// TwinCAT 3 PLC project LoggingHelper
// Title: Logging Helper
// Company: Beckhoff Industrial
// ProjectVersion: 0.1.0
// ProgramVersion: 3.1.4026.22
// libraries:
//   Tc2_Standard, * (Beckhoff Automation GmbH)
//   Tc2_System, * (Beckhoff Automation GmbH)
//   Tc2_Utilities, * (Beckhoff Automation GmbH)
// project tree:
//   Loggers/Interfaces/ I_LocalLogger.TcIO, I_Logger.TcIO
//   Loggers/ LocalLogger.TcPOU
//   LogMessages/Interfaces/ I_LogSource.TcIO, I_LogMessage.TcIO, I_LogArgument.TcIO
//   LogMessages/ LogMessage.TcPOU, LogSource.TcPOU
//   / Parameters.TcGVL, PlcTask.TcTTO
//   Project Information/ F_GetCompany.TcPOU, F_GetTitle.TcPOU, F_GetVersion.TcPOU
//   SimpleLogger/ I_LogPublisher.TcIO, LogHelper.TcPOU
//   Version/ Global_Version.TcGVL
//   _Internal/Interfaces/ I_Base.TcIO

CONFIGURATION LoggingHelper
    RESOURCE PLC ON TwinCAT3
        TASK PlcTask(INTERVAL := T#10ms, PRIORITY := 20);
    END_RESOURCE
END_CONFIGURATION

// ---- Parameters.TcGVL
{attribute 'qualified_only'}
VAR_GLOBAL CONSTANT
	MaxMessages : USINT := 10;
END_VAR

// ---- Version/Global_Version.TcGVL
{attribute 'TcGenerated'}
{attribute 'no-analysis'}
{attribute 'linkalways'}
// This function has been automatically generated from the project information.
VAR_GLOBAL CONSTANT
	{attribute 'const_non_replaced'}
	stLibVersion_Logging_Helper : ST_LibVersion := (iMajor := 0, iMinor := 1, iBuild := 0, iRevision := 0, nFlags := 0, sVersion := '0.1.0');
END_VAR

// ---- Loggers/Interfaces/I_LocalLogger.TcIO
INTERFACE I_LocalLogger EXTENDS I_Logger

METHOD ClearLog
VAR_INPUT
END_VAR
END_METHOD

{attribute 'monitoring' := 'call'}
PROPERTY Messages : REFERENCE TO ARRAY[0..Parameters.MaxMessages - 1] OF T_MaxString
GET
END_GET
END_PROPERTY

END_INTERFACE

// ---- Loggers/Interfaces/I_Logger.TcIO
INTERFACE I_Logger EXTENDS I_Base

METHOD LogMessage
VAR_INPUT
	Source	 : I_LogSource;
	Message	 : I_LogMessage;
	Argument : I_LogArgument := 0;
END_VAR
END_METHOD

END_INTERFACE

// ---- LogMessages/Interfaces/I_LogSource.TcIO
INTERFACE I_LogSource EXTENDS I_Base

{attribute 'monitoring':='call'}
PROPERTY SourceName : T_MaxString
GET
END_GET
END_PROPERTY

{attribute 'monitoring':='call'}
PROPERTY Timestamp : T_FILETIME64
GET
END_GET
END_PROPERTY

END_INTERFACE

// ---- LogMessages/Interfaces/I_LogMessage.TcIO
INTERFACE I_LogMessage EXTENDS I_Base

{attribute 'monitoring':='call'}
PROPERTY Message : T_MaxString
GET
END_GET
END_PROPERTY

{attribute 'monitoring':='call'}
PROPERTY Severity : USINT
GET
END_GET
END_PROPERTY

END_INTERFACE

// ---- LogMessages/Interfaces/I_LogArgument.TcIO
INTERFACE I_LogArgument EXTENDS I_Base

METHOD ToString : T_MaxString
VAR_INPUT
END_VAR
END_METHOD

END_INTERFACE

// ---- SimpleLogger/I_LogPublisher.TcIO
INTERFACE I_LogPublisher EXTENDS I_Base

METHOD Subscribe : BOOL
VAR_INPUT
	Logger : I_Logger;
END_VAR
END_METHOD

METHOD Unsubscribe : BOOL
VAR_INPUT
	Logger : I_Logger;
END_VAR
END_METHOD

END_INTERFACE

// ---- _Internal/Interfaces/I_Base.TcIO
INTERFACE I_Base EXTENDS SYSTEM.__QUERYINTERFACE

END_INTERFACE

// ---- Loggers/LocalLogger.TcPOU
FUNCTION_BLOCK LocalLogger IMPLEMENTS I_LocalLogger
VAR
	{attribute 'hide'}
	_Messages	 : ARRAY[0..Parameters.MaxMessages - 1] OF T_MaxString;
END_VAR

METHOD ClearLog
VAR_INPUT
END_VAR
VAR
	i : UDINT;
END_VAR
FOR i := 0 TO Parameters.MaxMessages - 1 DO
	_Messages[i] := '';
END_FOR
END_METHOD

METHOD LogMessage
VAR_INPUT
	Source	 : I_LogSource;
	Message	 : I_LogMessage;
	Argument : I_LogArgument := 0;
END_VAR

VAR
	TimeStamp  : T_FILETIME64;
	TimeString : T_MaxString;
	i : UDINT;
END_VAR
IF Source.TimeStamp = 0 THEN
	TimeStamp := F_GetSystemTime();
ELSE
	TimeStamp := Source.Timestamp;
END_IF

TimeString := SYSTEMTIME_TO_STRING(FILETIME64_TO_SYSTEMTIME(TimeStamp));
//shift messages down
FOR i := 2 TO Parameters.MaxMessages - 1 DO
	_Messages[Parameters.MaxMessages - i] := _Messages[Parameters.MaxMessages - 1 - i];
END_FOR

_Messages[0] := CONCAT(TimeString, CONCAT(' ', CONCAT(Source.SourceName, CONCAT(': ', Message.Message))));
IF Argument <> 0 THEN
	_Messages[0] := CONCAT(_Messages[0], CONCAT(' : ', Argument.ToString()));
END_IF
END_METHOD

{attribute 'monitoring' := 'call'}
PROPERTY Messages : REFERENCE TO ARRAY[0..Parameters.MaxMessages - 1] OF T_MaxString
GET
Messages REF= _Messages;
END_GET
END_PROPERTY

END_FUNCTION_BLOCK

// ---- LogMessages/LogMessage.TcPOU
FUNCTION_BLOCK LogMessage IMPLEMENTS I_LogMessage
VAR
	{attribute 'hide'}
	_Message : T_MaxString;
	{attribute 'hide'}
	_Severity : USINT;
END_VAR

{attribute 'monitoring':='call'}
PROPERTY Message : T_MaxString
GET
Message := _Message;
END_GET
SET
_Message := Message;
END_SET
END_PROPERTY

{attribute 'monitoring':='call'}
PROPERTY Severity : USINT
GET
Severity := _Severity;
END_GET
SET
_Severity := Severity;
END_SET
END_PROPERTY

END_FUNCTION_BLOCK

// ---- LogMessages/LogSource.TcPOU
FUNCTION_BLOCK LogSource IMPLEMENTS I_LogSource
VAR
	{attribute 'hide'}
	_SourceName : T_MaxString;
	{attribute 'hide'}
	_Timestamp : T_FILETIME64;
END_VAR

{attribute 'monitoring':='call'}
PROPERTY SourceName : T_MaxString
GET
Sourcename := _Sourcename;
END_GET
SET
_SourceName := SourceName;
END_SET
END_PROPERTY

{attribute 'monitoring':='call'}
PROPERTY Timestamp : T_FILETIME64
GET
Timestamp := _Timestamp;
END_GET
SET
_Timestamp := Timestamp;
END_SET
END_PROPERTY

END_FUNCTION_BLOCK

// ---- Project Information/F_GetCompany.TcPOU
// This function has been automatically generated from the project information.
{attribute 'signature_flag' := '1073741824'}
{attribute 'TcGenerated'}
{attribute 'no-analysis'}
FUNCTION F_GetCompany : WSTRING
VAR_INPUT
	
END_VAR

F_GetCompany := "Beckhoff Industrial";

END_FUNCTION

// ---- Project Information/F_GetTitle.TcPOU
// This function has been automatically generated from the project information.
{attribute 'signature_flag' := '1073741824'}
{attribute 'TcGenerated'}
{attribute 'no-analysis'}
FUNCTION F_GetTitle : WSTRING
VAR_INPUT
	
END_VAR

F_GetTitle := "Logging Helper";

END_FUNCTION

// ---- Project Information/F_GetVersion.TcPOU
// This function has been automatically generated from the project information.
{attribute 'signature_flag' := '1073741824'}
{attribute 'TcGenerated'}
{attribute 'no-analysis'}
FUNCTION F_GetVersion : ST_LibVersion
VAR_INPUT
	
END_VAR

F_GetVersion.iMajor := 0;
F_GetVersion.iMinor := 1;
F_GetVersion.iBuild := 0;
F_GetVersion.iRevision := 0;
F_GetVersion.sVersion := '0.1.0';
F_GetVersion.nFlags := 0;

END_FUNCTION

// ---- SimpleLogger/LogHelper.TcPOU
FUNCTION_BLOCK LogHelper
VAR_GENERIC CONSTANT
	MaxNumberOfSubscribers : USINT := 5;
END_VAR IMPLEMENTS I_LogPublisher
VAR
	SubscriberCount	   : USINT;
	_SubscribedLoggers : ARRAY[0..MaxNumberOfSubscribers - 1] OF I_Logger;
END_VAR

METHOD LogMessage
VAR_INPUT
	Source	 : I_LogSource;
	Message	 : I_LogMessage;
	Argument : I_LogArgument := 0;
END_VAR
VAR
	i : UDINT;
END_VAR
FOR i := 0 TO SubscriberCount - 1 DO
	IF _SubscribedLoggers[i] = 0 THEN
		//Don't create page faults with empty entries
		CONTINUE;
	END_IF

	//vary log calls depending on if there is an argument provided or not
	IF Argument = 0 THEN
		_SubscribedLoggers[i].LogMessage(Source := Source, Message := Message);
	ELSE
		_SubscribedLoggers[i].LogMessage(Source := Source, Message := Message, Argument := Argument);
	END_IF
END_FOR
END_METHOD

METHOD Subscribe : BOOL
VAR_INPUT
	Logger : I_Logger;
END_VAR
VAR
	i : UDINT;
END_VAR
IF SubscriberCount >= MaxNumberOfSubscribers THEN
	//Unable to accept any new loggers, early exit
	RETURN;
END_IF

FOR i := 0 TO MaxNumberOfSubscribers - 1 DO
	IF _SubscribedLoggers[i] = Logger THEN
		//Don't allow duplicates
		RETURN;
	END_IF

	IF _SubscribedLoggers[i] = 0 THEN
		//Add the logger , incremement count and return succcess
		_SubscribedLoggers[i] := Logger;
		SubscriberCount		  := SubscriberCount + 1;
		Subscribe			  := TRUE;
		RETURN;
	END_IF
END_FOR
END_METHOD

METHOD Unsubscribe : BOOL
VAR_INPUT
	Logger : I_Logger;
END_VAR

VAR
	i : USINT;
END_VAR
IF SubscriberCount = 0 THEN
	//Don't bother if no subscriptions are present
	RETURN;
END_IF

FOR i := 0 TO SubscriberCount - 1 DO
	IF _SubscribedLoggers[i] = 0 THEN
		//Don't do anything on empty log entries
		CONTINUE;
	END_IF

	IF _SubscribedLoggers[i] = Logger THEN
		//Remove logger, decrement and return true
		_SubScribedLoggers[i] := 0;
		SubscriberCount		  := SubscriberCount - 1;
		Unsubscribe			  := TRUE;
		RETURN;
	END_IF
END_FOR
END_METHOD

END_FUNCTION_BLOCK
